// TIA Portal V20 export
DATA_BLOCK "HmiInterface"   // DB81
// stored: Access Published, MemoryReserve 100, Namespace Unit1.Em1
   VAR
      em : "LAF_typeEmInterface";
      emHomedCheck : "Unit1.Em1.typeEmHomedCheck";
      cm { S7_SetPoint := 'True'} : "Unit1.Em1.typeCmInterface";
      unWinder : "LER_typeSequenceInterface";
   END_VAR
   VAR RETAIN
      cmUnWinderAxisB : "LBC_typeAxisControlInterface";
      cmAirShaftOnOff : "LBC_typeTwoWayActuatorInterface";
      cmExpelFwdBwd : "LBC_typeTwoWayActuatorInterface";
      cmTensionCheckSensor : "LBC_typeDigitalSignalInterface";
      cmRadiusMeasureAnalogInput : "LBC_typeAnalogInputInterface";
      cmEpc : "LER_typeCON600Interface";
      cmRadiusMeasure : "LER_typeRadiusMeasureInterface";
      cmUnWinderAxisB_TorqueCal : "LER_typeServoTorqueCalInterface";
      cmBobinID : "LER_typeRFIDInterface";
      cmEpc_UnUse : Bool;
      cmWinderDirectionChange : Bool := TRUE;
   END_VAR
   VAR
      AutoSpliceRemainingLength : LReal;
      SLS_EffectiveSpeed : LReal;
   END_VAR
BEGIN
   // cmBobinID.monitoring.error : RFID Error
END_DATA_BLOCK
